IF SUPER^.Step(980,TRUE,'Step number 980') THEN		
	SUPER^.StepCompleteWhen((_runOneStep OR _runAllSteps) AND _finishStep);	
	IF _runOneStep THEN	
		_runOneStep := FALSE;
		RETURN;
	END_IF	
END_IF		
		
IF SUPER^.Step(981,TRUE,'Step number 981') THEN		
	SUPER^.StepCompleteWhen((_runOneStep OR _runAllSteps) AND _finishStep);	
	IF _runOneStep THEN	
		_runOneStep := FALSE;
		RETURN;
	END_IF	
END_IF		
		
IF SUPER^.Step(982,TRUE,'Step number 982') THEN		
	SUPER^.StepCompleteWhen((_runOneStep OR _runAllSteps) AND _finishStep);	
	IF _runOneStep THEN	
		_runOneStep := FALSE;
		RETURN;
	END_IF	
END_IF		
		
IF SUPER^.Step(983,TRUE,'Step number 983') THEN		
	SUPER^.StepCompleteWhen((_runOneStep OR _runAllSteps) AND _finishStep);	
	IF _runOneStep THEN	
		_runOneStep := FALSE;
		RETURN;
	END_IF	
END_IF		
		
IF SUPER^.Step(984,TRUE,'Step number 984') THEN		
	SUPER^.StepCompleteWhen((_runOneStep OR _runAllSteps) AND _finishStep);	
	IF _runOneStep THEN	
		_runOneStep := FALSE;
		RETURN;
	END_IF	
END_IF		
		
IF SUPER^.Step(985,TRUE,'Step number 985') THEN		
	SUPER^.StepCompleteWhen((_runOneStep OR _runAllSteps) AND _finishStep);	
	IF _runOneStep THEN	
		_runOneStep := FALSE;
		RETURN;
	END_IF	
END_IF		
		
IF SUPER^.Step(986,TRUE,'Step number 986') THEN		
	SUPER^.StepCompleteWhen((_runOneStep OR _runAllSteps) AND _finishStep);	
	IF _runOneStep THEN	
		_runOneStep := FALSE;
		RETURN;
	END_IF	
END_IF		
		
IF SUPER^.Step(987,TRUE,'Step number 987') THEN		
	SUPER^.StepCompleteWhen((_runOneStep OR _runAllSteps) AND _finishStep);	
	IF _runOneStep THEN	
		_runOneStep := FALSE;
		RETURN;
	END_IF	
END_IF		
		
IF SUPER^.Step(988,TRUE,'Step number 988') THEN		
	SUPER^.StepCompleteWhen((_runOneStep OR _runAllSteps) AND _finishStep);	
	IF _runOneStep THEN	
		_runOneStep := FALSE;
		RETURN;
	END_IF	
END_IF		
		
IF SUPER^.Step(989,TRUE,'Step number 989') THEN		
	SUPER^.StepCompleteWhen((_runOneStep OR _runAllSteps) AND _finishStep);	
	IF _runOneStep THEN	
		_runOneStep := FALSE;
		RETURN;
	END_IF	
END_IF		
		
IF SUPER^.Step(990,TRUE,'Step number 990') THEN		
	SUPER^.StepCompleteWhen((_runOneStep OR _runAllSteps) AND _finishStep);	
	IF _runOneStep THEN	
		_runOneStep := FALSE;
		RETURN;
	END_IF	
END_IF		
		
IF SUPER^.Step(991,TRUE,'Step number 991') THEN		
	SUPER^.StepCompleteWhen((_runOneStep OR _runAllSteps) AND _finishStep);	
	IF _runOneStep THEN	
		_runOneStep := FALSE;
		RETURN;
	END_IF	
END_IF		
		
IF SUPER^.Step(992,TRUE,'Step number 992') THEN		
	SUPER^.StepCompleteWhen((_runOneStep OR _runAllSteps) AND _finishStep);	
	IF _runOneStep THEN	
		_runOneStep := FALSE;
		RETURN;
	END_IF	
END_IF		
		
IF SUPER^.Step(993,TRUE,'Step number 993') THEN		
	SUPER^.StepCompleteWhen((_runOneStep OR _runAllSteps) AND _finishStep);	
	IF _runOneStep THEN	
		_runOneStep := FALSE;
		RETURN;
	END_IF	
END_IF		
		
IF SUPER^.Step(994,TRUE,'Step number 994') THEN		
	SUPER^.StepCompleteWhen((_runOneStep OR _runAllSteps) AND _finishStep);	
	IF _runOneStep THEN	
		_runOneStep := FALSE;
		RETURN;
	END_IF	
END_IF		
		
IF SUPER^.Step(995,TRUE,'Step number 995') THEN		
	SUPER^.StepCompleteWhen((_runOneStep OR _runAllSteps) AND _finishStep);	
	IF _runOneStep THEN	
		_runOneStep := FALSE;
		RETURN;
	END_IF	
END_IF		
		
IF SUPER^.Step(996,TRUE,'Step number 996') THEN		
	SUPER^.StepCompleteWhen((_runOneStep OR _runAllSteps) AND _finishStep);	
	IF _runOneStep THEN	
		_runOneStep := FALSE;
		RETURN;
	END_IF	
END_IF		
		
IF SUPER^.Step(997,TRUE,'Step number 997') THEN		
	SUPER^.StepCompleteWhen((_runOneStep OR _runAllSteps) AND _finishStep);	
	IF _runOneStep THEN	
		_runOneStep := FALSE;
		RETURN;
	END_IF	
END_IF		
		
IF SUPER^.Step(998,TRUE,'Step number 998') THEN		
	SUPER^.StepCompleteWhen((_runOneStep OR _runAllSteps) AND _finishStep);	
	IF _runOneStep THEN	
		_runOneStep := FALSE;
		RETURN;
	END_IF	
END_IF		
		
IF SUPER^.Step(999,TRUE,'Step number 999') THEN		
	SUPER^.StepCompleteWhen((_runOneStep OR _runAllSteps) AND _finishStep);	
	IF _runOneStep THEN	
		_runOneStep := FALSE;
		RETURN;
	END_IF	
END_IF		
		
IF SUPER^.Step(1000,TRUE,'Step number 1000') THEN		
	SUPER^.StepCompleteWhen((_runOneStep OR _runAllSteps) AND _finishStep);	
	IF _runOneStep THEN	
		_runOneStep := FALSE;
		RETURN;
	END_IF	
END_IF		
		
IF SUPER^.Step(1001,TRUE,'Step number 1001') THEN		
	SUPER^.StepCompleteWhen((_runOneStep OR _runAllSteps) AND _finishStep);	
	IF _runOneStep THEN	
		_runOneStep := FALSE;
		RETURN;
	END_IF	
END_IF		
		
IF SUPER^.Step(1002,TRUE,'Step number 1002') THEN		
	SUPER^.StepCompleteWhen((_runOneStep OR _runAllSteps) AND _finishStep);	
	IF _runOneStep THEN	
		_runOneStep := FALSE;
		RETURN;
	END_IF	
END_IF		
		
IF SUPER^.Step(1003,TRUE,'Step number 1003') THEN		
	SUPER^.StepCompleteWhen((_runOneStep OR _runAllSteps) AND _finishStep);	
	IF _runOneStep THEN	
		_runOneStep := FALSE;
		RETURN;
	END_IF	
END_IF		
		
IF SUPER^.Step(1004,TRUE,'Step number 1004') THEN		
	SUPER^.StepCompleteWhen((_runOneStep OR _runAllSteps) AND _finishStep);	
	IF _runOneStep THEN	
		_runOneStep := FALSE;
		RETURN;
	END_IF	
END_IF		
		
IF SUPER^.Step(1005,TRUE,'Step number 1005') THEN		
	SUPER^.StepCompleteWhen((_runOneStep OR _runAllSteps) AND _finishStep);	
	IF _runOneStep THEN	
		_runOneStep := FALSE;
		RETURN;
	END_IF	
END_IF		
		
IF SUPER^.Step(1006,TRUE,'Step number 1006') THEN		
	SUPER^.StepCompleteWhen((_runOneStep OR _runAllSteps) AND _finishStep);	
	IF _runOneStep THEN	
		_runOneStep := FALSE;
		RETURN;
	END_IF	
END_IF		
		
IF SUPER^.Step(1007,TRUE,'Step number 1007') THEN		
	SUPER^.StepCompleteWhen((_runOneStep OR _runAllSteps) AND _finishStep);	
	IF _runOneStep THEN	
		_runOneStep := FALSE;
		RETURN;
	END_IF	
END_IF		
		
IF SUPER^.Step(1008,TRUE,'Step number 1008') THEN		
	SUPER^.StepCompleteWhen((_runOneStep OR _runAllSteps) AND _finishStep);	
	IF _runOneStep THEN	
		_runOneStep := FALSE;
		RETURN;
	END_IF	
END_IF		
		
IF SUPER^.Step(1009,TRUE,'Step number 1009') THEN		
	SUPER^.StepCompleteWhen((_runOneStep OR _runAllSteps) AND _finishStep);	
	IF _runOneStep THEN	
		_runOneStep := FALSE;
		RETURN;
	END_IF	
END_IF		
		
IF SUPER^.Step(1010,TRUE,'Step number 1010') THEN		
	SUPER^.StepCompleteWhen((_runOneStep OR _runAllSteps) AND _finishStep);	
	IF _runOneStep THEN	
		_runOneStep := FALSE;
		RETURN;
	END_IF	
END_IF		
		
IF SUPER^.Step(1011,TRUE,'Step number 1011') THEN		
	SUPER^.StepCompleteWhen((_runOneStep OR _runAllSteps) AND _finishStep);	
	IF _runOneStep THEN	
		_runOneStep := FALSE;
		RETURN;
	END_IF	
END_IF		
		
IF SUPER^.Step(1012,TRUE,'Step number 1012') THEN		
	SUPER^.StepCompleteWhen((_runOneStep OR _runAllSteps) AND _finishStep);	
	IF _runOneStep THEN	
		_runOneStep := FALSE;
		RETURN;
	END_IF	
END_IF		
		
IF SUPER^.Step(1013,TRUE,'Step number 1013') THEN		
	SUPER^.StepCompleteWhen((_runOneStep OR _runAllSteps) AND _finishStep);	
	IF _runOneStep THEN	
		_runOneStep := FALSE;
		RETURN;
	END_IF	
END_IF		
		
IF SUPER^.Step(1014,TRUE,'Step number 1014') THEN		
	SUPER^.StepCompleteWhen((_runOneStep OR _runAllSteps) AND _finishStep);	
	IF _runOneStep THEN	
		_runOneStep := FALSE;
		RETURN;
	END_IF	
END_IF		
		
IF SUPER^.Step(1015,TRUE,'Step number 1015') THEN		
	SUPER^.StepCompleteWhen((_runOneStep OR _runAllSteps) AND _finishStep);	
	IF _runOneStep THEN	
		_runOneStep := FALSE;
		RETURN;
	END_IF	
END_IF		
		
IF SUPER^.Step(1016,TRUE,'Step number 1016') THEN		
	SUPER^.StepCompleteWhen((_runOneStep OR _runAllSteps) AND _finishStep);	
	IF _runOneStep THEN	
		_runOneStep := FALSE;
		RETURN;
	END_IF	
END_IF		
		
IF SUPER^.Step(1017,TRUE,'Step number 1017') THEN		
	SUPER^.StepCompleteWhen((_runOneStep OR _runAllSteps) AND _finishStep);	
	IF _runOneStep THEN	
		_runOneStep := FALSE;
		RETURN;
	END_IF	
END_IF		
		
IF SUPER^.Step(1018,TRUE,'Step number 1018') THEN		
	SUPER^.StepCompleteWhen((_runOneStep OR _runAllSteps) AND _finishStep);	
	IF _runOneStep THEN	
		_runOneStep := FALSE;
		RETURN;
	END_IF	
END_IF		
		
IF SUPER^.Step(1019,TRUE,'Step number 1019') THEN		
	SUPER^.StepCompleteWhen((_runOneStep OR _runAllSteps) AND _finishStep);	
	IF _runOneStep THEN	
		_runOneStep := FALSE;
		RETURN;
	END_IF	
END_IF		
		
IF SUPER^.Step(1020,TRUE,'Step number 1020') THEN		
	SUPER^.StepCompleteWhen((_runOneStep OR _runAllSteps) AND _finishStep);	
	IF _runOneStep THEN	
		_runOneStep := FALSE;
		RETURN;
	END_IF	
END_IF		
		
IF SUPER^.Step(1021,TRUE,'Step number 1021') THEN		
	SUPER^.StepCompleteWhen((_runOneStep OR _runAllSteps) AND _finishStep);	
	IF _runOneStep THEN	
		_runOneStep := FALSE;
		RETURN;
	END_IF	
END_IF		
		
IF SUPER^.Step(1022,TRUE,'Step number 1022') THEN		
	SUPER^.StepCompleteWhen((_runOneStep OR _runAllSteps) AND _finishStep);	
	IF _runOneStep THEN	
		_runOneStep := FALSE;
		RETURN;
	END_IF	
END_IF		
		
IF SUPER^.Step(1023,TRUE,'Step number 1023') THEN		
	SUPER^.StepCompleteWhen((_runOneStep OR _runAllSteps) AND _finishStep);	
	IF _runOneStep THEN	
		_runOneStep := FALSE;
		RETURN;
	END_IF	
END_IF		
		
//******************************************************************
IF SUPER^.Step(_stepId,_enabled,_stepDescription) THEN
	SUPER^.StepCompleteWhen((_runOneStep OR _runAllSteps) AND _finishStep);	
	IF _runOneStep THEN	
		_runOneStep := FALSE;
		RETURN;
	END_IF		
END_IF
END_METHOD

METHOD PROTECTED OnSequenceCompleted
_onSequenceCompleteCount := _onSequenceCompleteCount + 1;
END_METHOD

METHOD PROTECTED OnSequencerError
VAR_INPUT
	inErrorId : eSequencerError;
END_VAR
CASE inErrorId OF
	eSequencerError.noError :
		_onSequencerErrorCount := _onSequencerErrorCount + 0;
	eSequencerError.NotUniqueStepId :
		_onSequencerErrorCount := _onSequencerErrorCount + 10;
	eSequencerError.StepIdHasBeenChanged :
		_onSequencerErrorCount := _onSequencerErrorCount + 20;
	eSequencerError.OrderOfTheStepHasBeenChanged :
		_onSequencerErrorCount := _onSequencerErrorCount + 40;
	eSequencerError.StepWithRequestedIdDoesNotExists :
		_onSequencerErrorCount := _onSequencerErrorCount + 50;
	eSequencerError.MultipleRequestStepMethodCall :
		_onSequencerErrorCount := _onSequencerErrorCount + 60;
	eSequencerError.StepIdTooLow :
		_onSequencerErrorCount := _onSequencerErrorCount + 70;
	eSequencerError.StepIdTooHigh :
		_onSequencerErrorCount := _onSequencerErrorCount + 80;
	ELSE
		_onSequencerErrorCount := _onSequencerErrorCount + 0;
END_CASE
END_METHOD

METHOD PROTECTED OnStateChange
VAR_INPUT
	PreviousState	: INT;
	NewState 		: INT;
END_VAR
THIS^._onStateChangeCount := THIS^._onStateChangeCount + 1;

_stateChangeFrom := PreviousState;
_stateChangeTo := NewState;

IF _callRestoreInOnStateChange THEN
	Restore();
END_IF
END_METHOD

METHOD PROTECTED OnStepCompleted
_onCompleteStepCount := _onCompleteStepCount + 1;
END_METHOD

PROPERTY INTERNAL RequestStepCycle : UINT
GET
RequestStepCycle := _requestStepCycle;
END_GET
SET
_requestStepCycle := RequestStepCycle;
END_SET
END_PROPERTY

METHOD INTERNAL SequencerClose
SUPER^._Close();
END_METHOD

METHOD INTERNAL SequencerHasError : BOOL
SequencerHasError := SUPER^._sequencerHasError;
END_METHOD

METHOD INTERNAL SequencerOpen
SUPER^._Open();
END_METHOD

METHOD INTERNAL SetChildState 
VAR_INPUT
	inState			:	INT;
END_VAR
THIS^._myTcoState.ChangeState(inState);
END_METHOD

METHOD INTERNAL SetCurrentStep 
VAR_INPUT
	inStepID 			:	INT;
	inStepDescription	:	STRING(254);
END_VAR
THIS^._currentStep.ID			:=	inStepID;
THIS^._currentStep.Description	:=	inStepDescription;
END_METHOD

METHOD SetCurrentStepToErrorState : BOOL
_currentStep.Status := TcoCore.eStepStatus.Error;

SetCurrentStepToErrorState := _currentStep.Status = TcoCore.eStepStatus.Error;
END_METHOD

METHOD SetCyclicMode : BOOL
ModeController.Mode := eSequencerMode.CyclicMode;

SetCyclicMode := ModeController.Mode = eSequencerMode.CyclicMode;
END_METHOD

METHOD SetInvalidMode : BOOL
ModeController.Mode := eSequencerMode.Invalid;

SetInvalidMode := ModeController.Mode = eSequencerMode.Invalid;
END_METHOD

METHOD INTERNAL SetNumberOfSteps 
VAR_INPUT
	inNumberOfSteps : UINT;
END_VAR
_stepCounter 						:=	inNumberOfSteps;
_numberOfStepsInSequence			:=	inNumberOfSteps;
_previousNumberOfStepsInSequence 	:=	inNumberOfSteps;
END_METHOD

METHOD INTERNAL SetSequenceAsChecked
_stepIDUniquenessChecked := TRUE;
_StepIdUniquenessState := eStepIdUniquenessState.Done;
END_METHOD

METHOD INTERNAL SetSequenceAsNotChecked
_stepIDUniquenessChecked := FALSE;
_StepIdUniquenessState := eStepIdUniquenessState.NotYetStarted;
END_METHOD

METHOD SetStepMode : BOOL
ModeController.Mode := eSequencerMode.StepMode;

SetStepMode := ModeController.Mode = eSequencerMode.StepMode;
END_METHOD

METHOD INTERNAL SetTestParams
VAR_INPUT
	inRunOneStep		:	BOOL;
	inRunAllSteps		:	BOOL;
	inFinishStep		:	BOOL;
	inID				:	UINT;
	inEnabled			:	BOOL;
	inStepDescription	:	STRING(254);	
END_VAR
THIS^._runOneStep		:=			inRunOneStep;
THIS^._runAllSteps 		:= 			inRunAllSteps;
THIS^._finishStep 		:= 			inFinishStep;
THIS^._stepId 				:=			inID;
THIS^._enabled 			:= 			inEnabled;
THIS^._stepDescription 	:=			inStepDescription;
END_METHOD

METHOD StepCount 
VAR_INPUT
    inTotalStepNumber : UINT;
    inFinishStep : BOOL;
END_VAR
VAR 
	i : INT;
	_lastStepId : INT;
END_VAR
FOR i:=0 TO inTotalStepNumber DO
	IF SUPER^.Step(i,TRUE,CONCAT('Step number ',INT_TO_STRING(i))) THEN		
		SUPER^.StepCompleteWhen(inFinishStep);	
	END_IF	
END_FOR
END_METHOD

{attribute 'TcRpcEnable'}
METHOD INTERNAL UpdateCurrentStepDetails
_currentStepId				:=	SUPER^._currentStep.ID;
_currentStepOrder			:=	SUPER^._currentStep.Order;
_currentStepEnabled			:=	SUPER^._currentStep.Enabled;
_currentStepDescription		:=	SUPER^._currentStep.Description;
_currentStepStatus			:=	SUPER^._currentStep.Status;
_currentStepDuration		:=	SUPER^._currentStep.Duration;
END_METHOD

END_FUNCTION_BLOCK

(* stored: Version 1.1.0.1
   POU _TcoSequence: Id {571e2ee4-f5b5-02ce-211f-57bbdaa7b236}, SpecialFunc None
   Folder _Tests: Id {fececb69-8a6c-070a-00eb-cef13c42f29f}
   Method _RequestStep: Id {f945a046-4478-0e84-16fe-f8bd6b886450}
   Method _RunExecutionSubstitute: Id {b4bf6879-f257-0cef-3de1-77387a9b129b}
   Method _SequenceComplete: Id {76fa3e54-f0d3-0ab3-25bb-7fddc5d6c99a}
   Method _Step: Id {0476214f-c22c-0ae2-289b-5585879fc253}
   Method _StepBackward: Id {75b5bd54-dbc4-0be2-0654-0e35a8d1a98c}
   Method _StepCompleteWhen: Id {f251b76e-e67d-01a9-1a7b-81f2a404f77b}
   Method _StepForward: Id {206d15c0-fe83-05d6-0ec6-db1186606838}
   Method _StepIn: Id {86d67c04-df8b-05e6-300a-20087f7700a3}
   Method ChildHasAutoRestoreEnabled: Id {c79fc47b-b084-00d5-293f-d922936eb0aa}
   Method ChildIsAutoRestorable: Id {e22dcdd0-bfe9-0535-1dc5-314880dadab4}
   Method CleanupPointers: Id {8003d78a-9184-09d1-09c6-aaadf42db71b}
   Method ClearNumberOfSteps: Id {9b33e6b0-198c-0edb-144d-61e1b7f0cab5}
   Method GetChildState: Id {2927dd52-15a1-0dd1-3c7d-097a40c1e561}
   Method GetNumberOfStepsInSequence: Id {88701eef-6787-0393-165a-e2a171e7efcc}
   Method GetSequencerErrorId: Id {914a46e2-3b46-0070-0ee0-2384096f76ba}
   Method GetTextOfTheMostImportantMessage: Id {41a8dd6c-ed7c-0f1c-07f3-045a2b8a8075}
   Method HasAutoRestoreEnabled: Id {e673c8ef-8c2e-02b5-0bfb-81a2eea94118}
   Method IsAutoRestorable: Id {73c86ef5-315c-03de-10c7-666548cfa304}
   Method IsFirstStepEntry: Id {ecb1f5e5-b132-06eb-3789-fbbee541f8c1}
   Method Main: Id {dfa40309-5ef0-0c33-3509-75275eb9f222}
   Method OnSequenceCompleted: Id {9e48380f-6fa1-0276-0d16-9cff2a551b24}
   Method OnSequencerError: Id {e60f61c0-19a7-09ab-1358-93f066a796d0}
   Method OnStateChange: Id {4b9ac3ba-15ad-09e4-1047-49ffade5bf2f}
   Method OnStepCompleted: Id {28a3607e-c2b1-05b1-1f50-2dc419501a6d}
   Property RequestStepCycle: Id {0b38355d-b804-0298-10a9-ed9778d81078}
   Get Get: Id {3394497e-91e5-057b-0e2c-1d00e5b238c3}
   Set Set: Id {578dd97e-2b21-01ee-19a3-3d007df7b986}
   Method SequencerClose: Id {0ad2e2a9-a9c5-094d-000e-7ba918276451}
   Method SequencerHasError: Id {261f1997-a645-0ecb-3f28-074af404a3f1}
   Method SequencerOpen: Id {1089978b-87c8-0b12-307b-f6cb0ea0de6b}
   Method SetChildState: Id {faa8995f-b5f8-02d8-38a3-2a613a630a27}
   Method SetCurrentStep: Id {715009f7-0632-0b33-2e9f-a5e2128be37a}
   Method SetCurrentStepToErrorState: Id {5f8d43a3-611c-0a6e-002b-06aa8a6cbe29}
   Method SetCyclicMode: Id {d3cc8daf-a03f-05bb-177c-e3e8d9f3a6f6}
   Method SetInvalidMode: Id {74b9d16f-d305-02e5-0970-ca5acfe60101}
   Method SetNumberOfSteps: Id {a6aa68df-90d7-0070-3c97-e0fbd1496a81}
   Method SetSequenceAsChecked: Id {dc8ac25e-7945-00b2-2e3f-3727febacee0}
   Method SetSequenceAsNotChecked: Id {7d667e47-1b17-06c5-1cbf-126f69b6422e}
   Method SetStepMode: Id {2b1583e6-8447-07dd-00c7-e876e9da521f}
   Method SetTestParams: Id {940b02ab-f027-07d6-277b-cd452ddc4de2}
   Method StepCount: Id {c228bb20-df6c-0702-0351-4c80a8280411}
   Method UpdateCurrentStepDetails: Id {a126d46a-827e-0f20-2f04-b588ce9b347a} *)
